PROGRAM Circuito_L1
VAR_INPUT
	Modo_Calibrar_L1: BOOL;
END_VAR

VAR
	fbLavado_L1 :LavadoCircuitoLiquidos;
	bhs :BOOL;
	rhs :REAL;
	ihs :INT;
	whs :WORD;
	ths :TIME;
	fbBomba_L1 :Equipo_Motor_ATV320;
	Totalizador_L1: Totalizador;
	Reset_TotL1:BOOL;
	ControlValv_ioLink_V1: ControlValv_ioLink;
	ControlValv_ioLink_V2: ControlValv_ioLink;
	ControlValv_ioLink_V3: ControlValv_ioLink;
	ControlValv_ioLink_V4: ControlValv_ioLink;
	Falla_L1_V1:BOOL;
	Falla_L1_V2:BOOL;
	Falla_L1_V3:BOOL;
	Falla_L1_V4:BOOL;
	Balanza_PU1_WT1: Balanza;
	dHS:DINT;
	TOF_calibradoIBC: TOF;
	TDemoraInyectar: TON;
	SetDemoraInyeccion: REAL;
	Volumen_L1: REAL;
	AuxVol: REAL;
	Total: REAL;
	auxIniCal: BOOL;
	Calculo_caudal_L1: Calculo_caudal;
	PID_L1_SP: REAL;
	PID_L1_PV: REAL;
	CorrecionCaudalxOffset_L1: CorrecionCaudalxOffset;
	tInyeccion: TON;
	PID_L1_manual: REAL;
	PID_L1: FB_PID;
	PID_L1_Kp: REAL := 0.1;
	PID_L1_Ti: REAL := 100;
	PID_L1_auto: BOOL;
	PID_L1_reset: BOOL;
	PID_L1_bMuerta: REAL := 5;
	Tiempo_seg_to_TIME_DemoraInyec: Tiempo_seg_to_TIME;
	AuxTDemoraInyec: TIME;
	Tiempo_TIME_to_seg_InyCal: Tiempo_TIME_to_seg;
	AuxInyCal:TIME;
	ProductoAsociado:STRING;
	Lavagem_Circuito01: Lavagem;
	RTRIG: ARRAY[1..10] OF R_TRIG;
	FiltroTeste: Filtro2;
END_VAR	
VAR PERSISTENT
	UltimaCalibracao	:UDINT;	//Data e hora da ultima calibração
END_VAR
VAR // added by the converter: edge detectors and wires of the graphical bodies
    _w1, _w2, _w3, _w4, _w5, _w6, _w7, _w8, _w9, _w10, _w11, _w12 : BOOL;
    _ft1 : F_TRIG;
    _rt1 : R_TRIG;
END_VAR

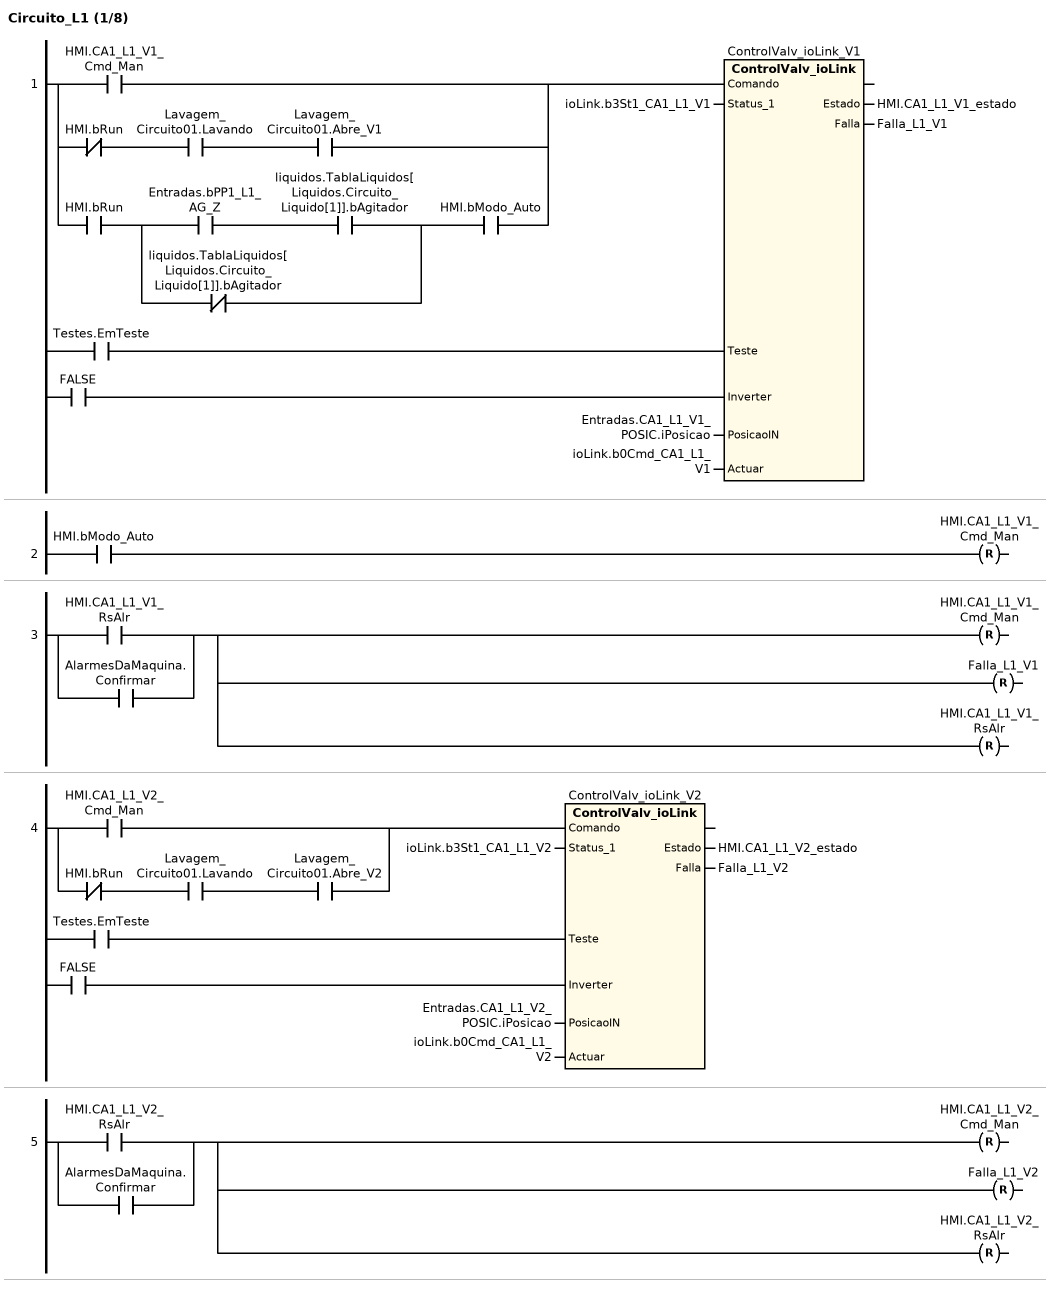
// NETWORK 1
ControlValv_ioLink_V1(
    Comando := HMI.CA1_L1_V1_Cmd_Man OR NOT HMI.bRun AND Lavagem_Circuito01.Lavando AND Lavagem_Circuito01.Abre_V1 OR HMI.bRun AND (Entradas.bPP1_L1_AG_Z AND (liquidos.TablaLiquidos[Liquidos.Circuito_Liquido[1]].bAgitador) OR NOT (liquidos.TablaLiquidos[Liquidos.Circuito_Liquido[1]].bAgitador)) AND HMI.bModo_Auto,
    Status_1 := ioLink.b3St1_CA1_L1_V1,
    Teste := Testes.EmTeste,
    Inverter := FALSE,
    PosicaoIN := Entradas.CA1_L1_V1_POSIC.iPosicao,
    Actuar := ioLink.b0Cmd_CA1_L1_V1,
    Estado => HMI.CA1_L1_V1_estado,
    Falla => Falla_L1_V1); // ControlValv_ioLink

// NETWORK 2
HMI.CA1_L1_V1_Cmd_Man R= HMI.bModo_Auto;

// NETWORK 3
_w1 := HMI.CA1_L1_V1_RsAlr OR AlarmesDaMaquina.Confirmar;
HMI.CA1_L1_V1_Cmd_Man R= _w1;
Falla_L1_V1 R= _w1;
HMI.CA1_L1_V1_RsAlr R= _w1;

// NETWORK 4
ControlValv_ioLink_V2(
    Comando := HMI.CA1_L1_V2_Cmd_Man OR NOT HMI.bRun AND Lavagem_Circuito01.Lavando AND Lavagem_Circuito01.Abre_V2,
    Status_1 := ioLink.b3St1_CA1_L1_V2,
    Teste := Testes.EmTeste,
    Inverter := FALSE,
    PosicaoIN := Entradas.CA1_L1_V2_POSIC.iPosicao,
    Actuar := ioLink.b0Cmd_CA1_L1_V2,
    Estado => HMI.CA1_L1_V2_estado,
    Falla => Falla_L1_V2); // ControlValv_ioLink

// NETWORK 5
_w2 := HMI.CA1_L1_V2_RsAlr OR AlarmesDaMaquina.Confirmar;
HMI.CA1_L1_V2_Cmd_Man R= _w2;
Falla_L1_V2 R= _w2;
HMI.CA1_L1_V2_RsAlr R= _w2;

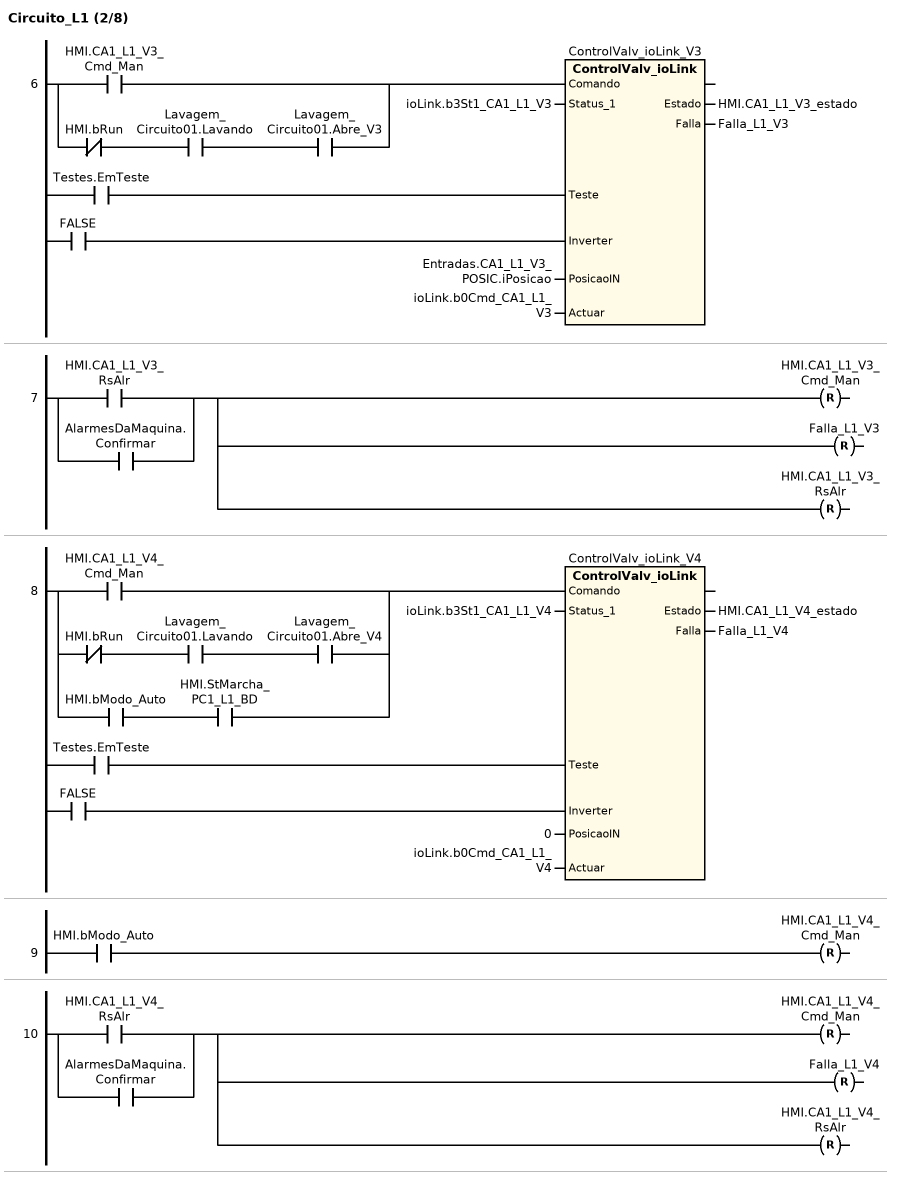
// NETWORK 6
ControlValv_ioLink_V3(
    Comando := HMI.CA1_L1_V3_Cmd_Man OR NOT HMI.bRun AND Lavagem_Circuito01.Lavando AND Lavagem_Circuito01.Abre_V3,
    Status_1 := ioLink.b3St1_CA1_L1_V3,
    Teste := Testes.EmTeste,
    Inverter := FALSE,
    PosicaoIN := Entradas.CA1_L1_V3_POSIC.iPosicao,
    Actuar := ioLink.b0Cmd_CA1_L1_V3,
    Estado => HMI.CA1_L1_V3_estado,
    Falla => Falla_L1_V3); // ControlValv_ioLink

// NETWORK 7
_w3 := HMI.CA1_L1_V3_RsAlr OR AlarmesDaMaquina.Confirmar;
HMI.CA1_L1_V3_Cmd_Man R= _w3;
Falla_L1_V3 R= _w3;
HMI.CA1_L1_V3_RsAlr R= _w3;

// NETWORK 8
ControlValv_ioLink_V4(
    Comando := HMI.CA1_L1_V4_Cmd_Man OR NOT HMI.bRun AND Lavagem_Circuito01.Lavando AND Lavagem_Circuito01.Abre_V4 OR HMI.bModo_Auto AND HMI.StMarcha_PC1_L1_BD,
    Status_1 := ioLink.b3St1_CA1_L1_V4,
    Teste := Testes.EmTeste,
    Inverter := FALSE,
    PosicaoIN := 0,
    Actuar := ioLink.b0Cmd_CA1_L1_V4,
    Estado => HMI.CA1_L1_V4_estado,
    Falla => Falla_L1_V4); // ControlValv_ioLink

// NETWORK 9
HMI.CA1_L1_V4_Cmd_Man R= HMI.bModo_Auto;

// NETWORK 10
_w4 := HMI.CA1_L1_V4_RsAlr OR AlarmesDaMaquina.Confirmar;
HMI.CA1_L1_V4_Cmd_Man R= _w4;
Falla_L1_V4 R= _w4;
HMI.CA1_L1_V4_RsAlr R= _w4;

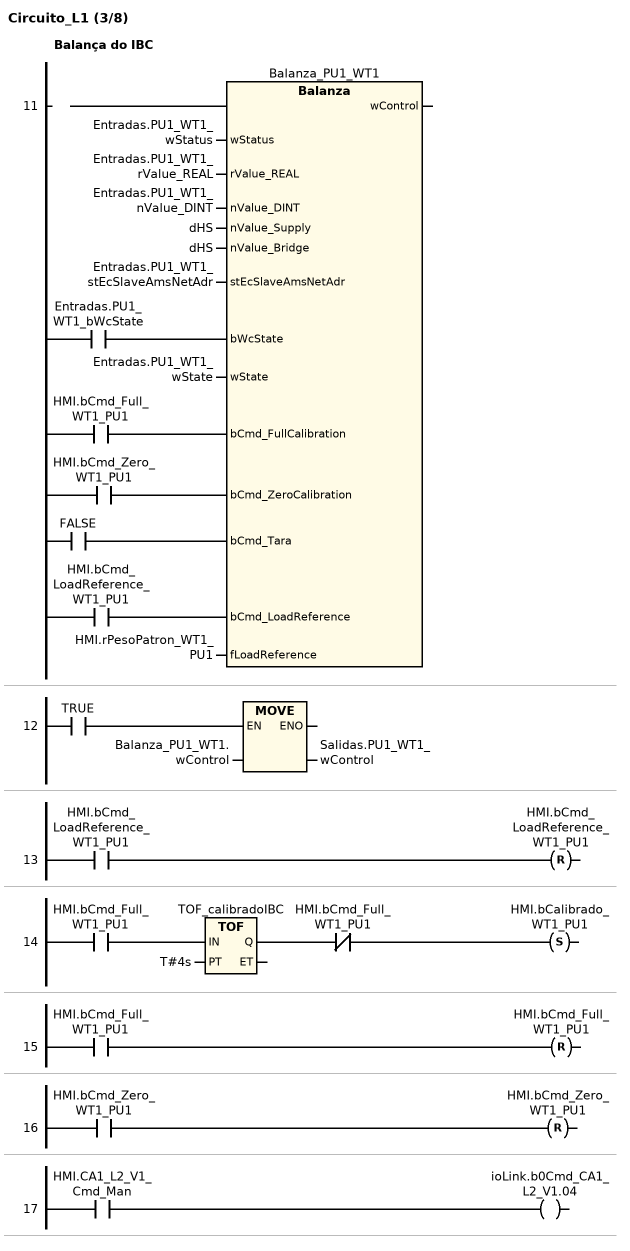
// NETWORK 11: Balança do IBC
Balanza_PU1_WT1(
    wStatus := Entradas.PU1_WT1_wStatus,
    rValue_REAL := Entradas.PU1_WT1_rValue_REAL,
    nValue_DINT := Entradas.PU1_WT1_nValue_DINT,
    nValue_Supply := dHS,
    nValue_Bridge := dHS,
    stEcSlaveAmsNetAdr := Entradas.PU1_WT1_stEcSlaveAmsNetAdr,
    bWcState := Entradas.PU1_WT1_bWcState,
    wState := Entradas.PU1_WT1_wState,
    bCmd_FullCalibration := HMI.bCmd_Full_WT1_PU1,
    bCmd_ZeroCalibration := HMI.bCmd_Zero_WT1_PU1,
    bCmd_Tara := FALSE,
    bCmd_LoadReference := HMI.bCmd_LoadReference_WT1_PU1,
    fLoadReference := HMI.rPesoPatron_WT1_PU1); // Balanza

// NETWORK 12
Salidas.PU1_WT1_wControl := Balanza_PU1_WT1.wControl;

// NETWORK 13
HMI.bCmd_LoadReference_WT1_PU1 R= HMI.bCmd_LoadReference_WT1_PU1;

// NETWORK 14
TOF_calibradoIBC(IN := HMI.bCmd_Full_WT1_PU1, PT := T#4s); // TOF
HMI.bCalibrado_WT1_PU1 S= TOF_calibradoIBC.Q AND NOT HMI.bCmd_Full_WT1_PU1;

// NETWORK 15
HMI.bCmd_Full_WT1_PU1 R= HMI.bCmd_Full_WT1_PU1;

// NETWORK 16
HMI.bCmd_Zero_WT1_PU1 R= HMI.bCmd_Zero_WT1_PU1;

// NETWORK 17
ioLink.b0Cmd_CA1_L2_V1.04 := HMI.CA1_L2_V1_Cmd_Man;

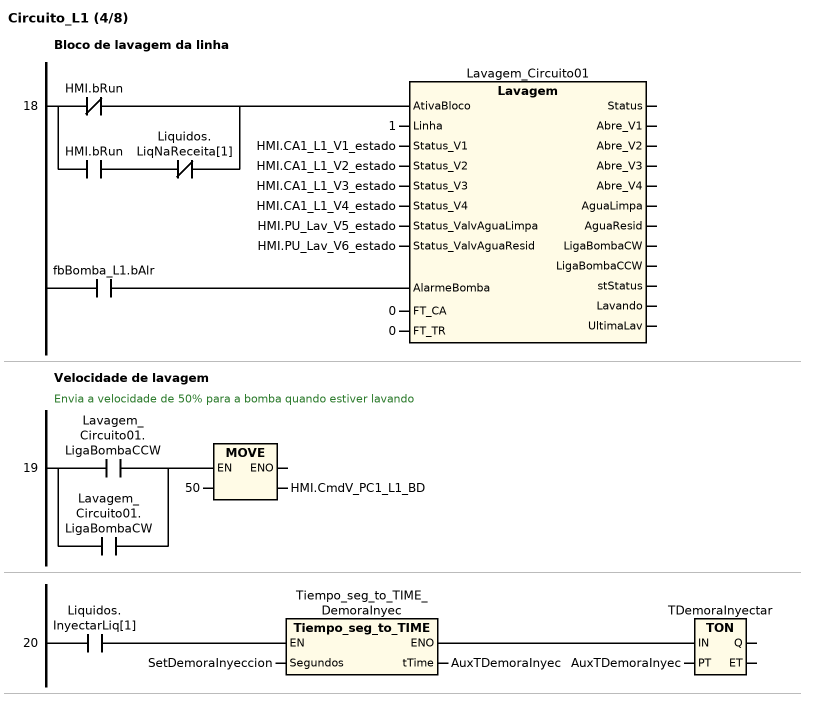
// NETWORK 18: Bloco de lavagem da linha
Lavagem_Circuito01(
    AtivaBloco := NOT HMI.bRun OR HMI.bRun AND NOT Liquidos.LiqNaReceita[1],
    Linha := 1,
    Status_V1 := HMI.CA1_L1_V1_estado,
    Status_V2 := HMI.CA1_L1_V2_estado,
    Status_V3 := HMI.CA1_L1_V3_estado,
    Status_V4 := HMI.CA1_L1_V4_estado,
    Status_ValvAguaLimpa := HMI.PU_Lav_V5_estado,
    Status_ValvAguaResid := HMI.PU_Lav_V6_estado,
    AlarmeBomba := fbBomba_L1.bAlr,
    FT_CA := 0,
    FT_TR := 0); // Lavagem

// NETWORK 19: Velocidade de lavagem
// Envia a velocidade de 50% para a bomba quando estiver lavando
IF Lavagem_Circuito01.LigaBombaCCW OR Lavagem_Circuito01.LigaBombaCW THEN HMI.CmdV_PC1_L1_BD := 50; END_IF

// NETWORK 20
_w5 := Liquidos.InyectarLiq[1];
IF _w5 THEN
    Tiempo_seg_to_TIME_DemoraInyec(Segundos := SetDemoraInyeccion, tTime => AuxTDemoraInyec); // Tiempo_seg_to_TIME
END_IF
TDemoraInyectar(IN := _w5, PT := AuxTDemoraInyec); // TON

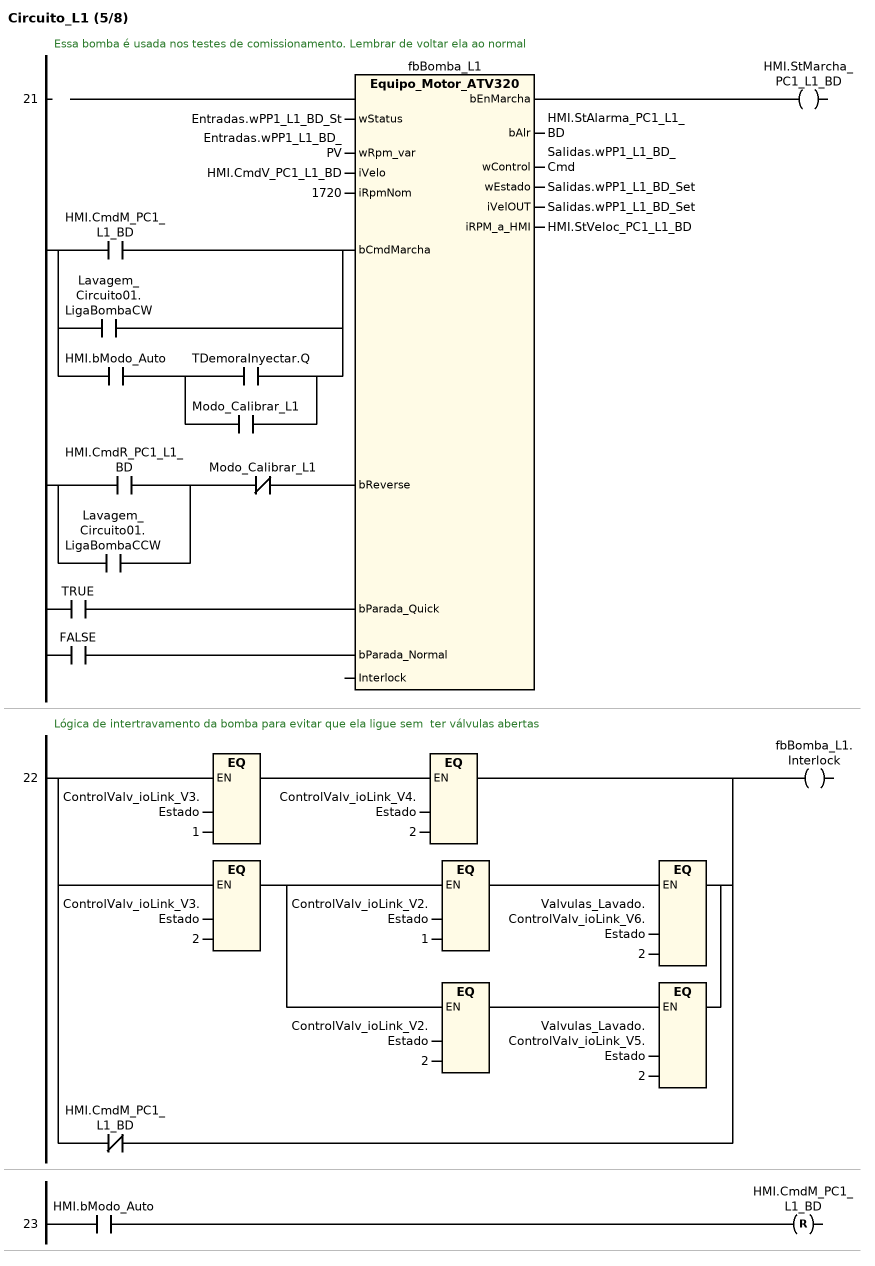
// NETWORK 21
// Essa bomba é usada nos testes de comissionamento. Lembrar de voltar ela ao normal
fbBomba_L1(
    wStatus := Entradas.wPP1_L1_BD_St,
    wRpm_var := Entradas.wPP1_L1_BD_PV,
    iVelo := HMI.CmdV_PC1_L1_BD,
    iRpmNom := 1720,
    bCmdMarcha := HMI.CmdM_PC1_L1_BD OR Lavagem_Circuito01.LigaBombaCW OR HMI.bModo_Auto AND (TDemoraInyectar.Q OR Modo_Calibrar_L1),
    bReverse := (HMI.CmdR_PC1_L1_BD OR Lavagem_Circuito01.LigaBombaCCW) AND NOT Modo_Calibrar_L1,
    bParada_Quick := TRUE,
    bParada_Normal := FALSE,
    bAlr => HMI.StAlarma_PC1_L1_BD,
    wControl => Salidas.wPP1_L1_BD_Cmd,
    wEstado => Salidas.wPP1_L1_BD_Set,
    iVelOUT => Salidas.wPP1_L1_BD_Set,
    iRPM_a_HMI => HMI.StVeloc_PC1_L1_BD); // Equipo_Motor_ATV320
HMI.StMarcha_PC1_L1_BD := fbBomba_L1.bEnMarcha;

// NETWORK 22
// Lógica de intertravamento da bomba para evitar que ela ligue sem  ter válvulas abertas
_w6 := NOT HMI.CmdM_PC1_L1_BD;
IF NOT _w6 THEN
    _w7 := ControlValv_ioLink_V3.Estado = 2;
    _w6 := ControlValv_ioLink_V3.Estado = 1 AND ControlValv_ioLink_V4.Estado = 2 OR (_w7 AND ControlValv_ioLink_V2.Estado = 1 AND Valvulas_Lavado.ControlValv_ioLink_V6.Estado = 2 OR _w7 AND ControlValv_ioLink_V2.Estado = 2 AND Valvulas_Lavado.ControlValv_ioLink_V5.Estado = 2);
END_IF
fbBomba_L1.Interlock := _w6;

// NETWORK 23
HMI.CmdM_PC1_L1_BD R= HMI.bModo_Auto;

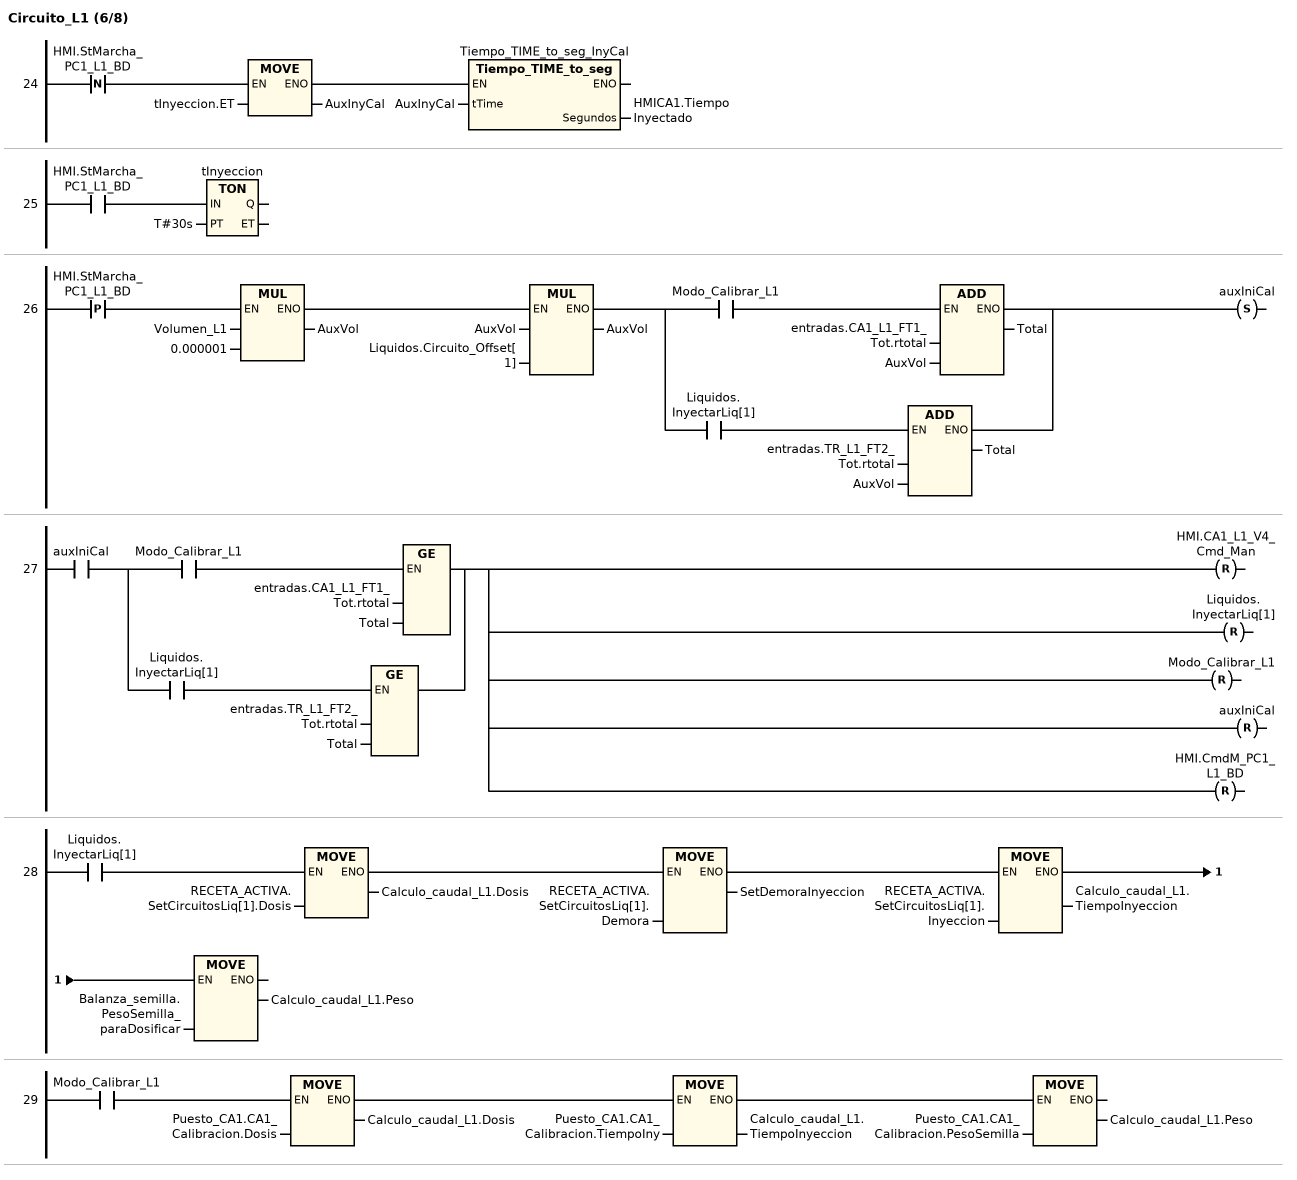
// NETWORK 24
_ft1(CLK := HMI.StMarcha_PC1_L1_BD);
_w8 := _ft1.Q;
IF _w8 THEN AuxInyCal := tInyeccion.ET; END_IF
IF _w8 THEN
    Tiempo_TIME_to_seg_InyCal(tTime := AuxInyCal, Segundos => HMICA1.TiempoInyectado); // Tiempo_TIME_to_seg
END_IF

// NETWORK 25
tInyeccion(IN := HMI.StMarcha_PC1_L1_BD, PT := T#30s); // TON

// NETWORK 26
_rt1(CLK := HMI.StMarcha_PC1_L1_BD);
_w9 := _rt1.Q;
IF _w9 THEN AuxVol := Volumen_L1 * 0.000001; END_IF
IF _w9 THEN AuxVol := AuxVol * Liquidos.Circuito_Offset[1]; END_IF
IF _w9 AND Modo_Calibrar_L1 THEN Total := entradas.CA1_L1_FT1_Tot.rtotal + AuxVol; END_IF
IF _w9 AND Liquidos.InyectarLiq[1] THEN Total := entradas.TR_L1_FT2_Tot.rtotal + AuxVol; END_IF
auxIniCal S= _w9 AND Modo_Calibrar_L1 OR _w9 AND Liquidos.InyectarLiq[1];

// NETWORK 27
_w10 := auxIniCal AND Modo_Calibrar_L1 AND entradas.CA1_L1_FT1_Tot.rtotal >= Total OR auxIniCal AND Liquidos.InyectarLiq[1] AND entradas.TR_L1_FT2_Tot.rtotal >= Total;
HMI.CA1_L1_V4_Cmd_Man R= _w10;
Liquidos.InyectarLiq[1] R= _w10;
Modo_Calibrar_L1 R= _w10;
auxIniCal R= _w10;
HMI.CmdM_PC1_L1_BD R= _w10;

// NETWORK 28
_w11 := Liquidos.InyectarLiq[1];
IF _w11 THEN Calculo_caudal_L1.Dosis := RECETA_ACTIVA.SetCircuitosLiq[1].Dosis; END_IF
IF _w11 THEN SetDemoraInyeccion := RECETA_ACTIVA.SetCircuitosLiq[1].Demora; END_IF
IF _w11 THEN Calculo_caudal_L1.TiempoInyeccion := RECETA_ACTIVA.SetCircuitosLiq[1].Inyeccion; END_IF
IF _w11 THEN Calculo_caudal_L1.Peso := Balanza_semilla.PesoSemilla_paraDosificar; END_IF

// NETWORK 29
_w12 := Modo_Calibrar_L1;
IF _w12 THEN Calculo_caudal_L1.Dosis := Puesto_CA1.CA1_Calibracion.Dosis; END_IF
IF _w12 THEN Calculo_caudal_L1.TiempoInyeccion := Puesto_CA1.CA1_Calibracion.TiempoIny; END_IF
IF _w12 THEN Calculo_caudal_L1.Peso := Puesto_CA1.CA1_Calibracion.PesoSemilla; END_IF

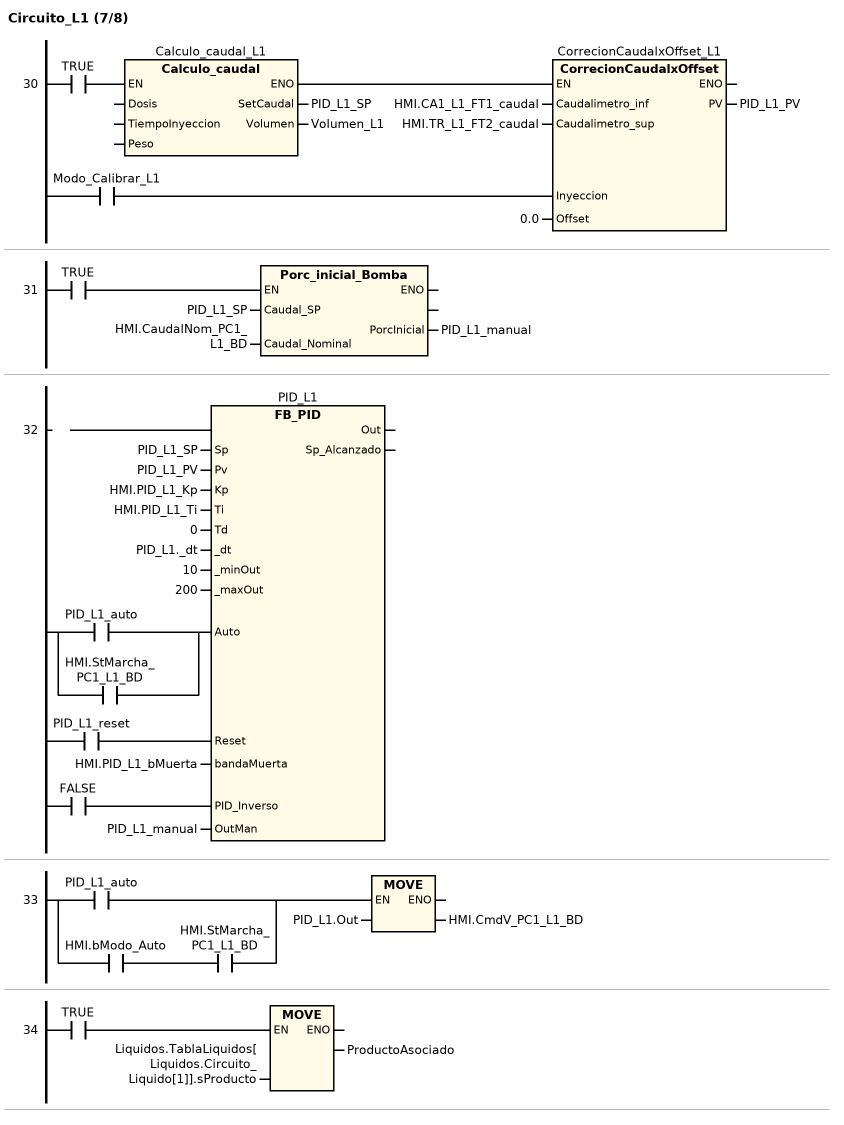
// NETWORK 30
Calculo_caudal_L1(SetCaudal => PID_L1_SP, Volumen => Volumen_L1); // Calculo_caudal
CorrecionCaudalxOffset_L1(
    Caudalimetro_inf := HMI.CA1_L1_FT1_caudal,
    Caudalimetro_sup := HMI.TR_L1_FT2_caudal,
    Inyeccion := Modo_Calibrar_L1,
    Offset := 0.0,
    PV => PID_L1_PV); // CorrecionCaudalxOffset

// NETWORK 31
Porc_inicial_Bomba(Caudal_SP := PID_L1_SP, Caudal_Nominal := HMI.CaudalNom_PC1_L1_BD, PorcInicial => PID_L1_manual);

// NETWORK 32
PID_L1(
    Sp := PID_L1_SP,
    Pv := PID_L1_PV,
    Kp := HMI.PID_L1_Kp,
    Ti := HMI.PID_L1_Ti,
    Td := 0,
    _dt := PID_L1._dt,
    _minOut := 10,
    _maxOut := 200,
    Auto := PID_L1_auto OR HMI.StMarcha_PC1_L1_BD,
    Reset := PID_L1_reset,
    bandaMuerta := HMI.PID_L1_bMuerta,
    PID_Inverso := FALSE,
    OutMan := PID_L1_manual); // FB_PID

// NETWORK 33
IF PID_L1_auto OR HMI.bModo_Auto AND HMI.StMarcha_PC1_L1_BD THEN HMI.CmdV_PC1_L1_BD := PID_L1.Out; END_IF

// NETWORK 34
ProductoAsociado := Liquidos.TablaLiquidos[Liquidos.Circuito_Liquido[1]].sProducto;

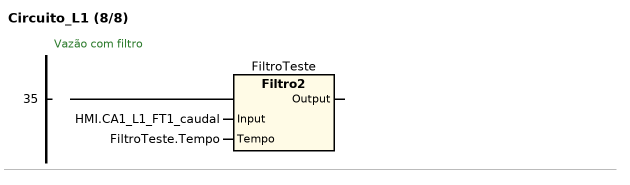
// NETWORK 35
// Vazão com filtro
FiltroTeste(Input := HMI.CA1_L1_FT1_caudal, Tempo := FiltroTeste.Tempo); // Filtro2

END_PROGRAM

(* stored: Version 1.1.0.1, ProductVersion 3.1.4024.14
   POU Circuito_L1: Id {771c4770-cd68-4ff4-98f9-2f0bc020eee1}, SpecialFunc None *)
